// TIA Portal project "Project3" (V15.1)

(* hardware
DEVICE "S7-1200 station_1"  S7-1200 Station
   slot 0: "Rack_0"  S7-1200 Rack  Rack  V1.0
   slot 1: "PLC_1"  CPU 1214C DC/DC/Rly  6ES7 214-1HG40-0XB0  V4.2
*)

// ===== PLC "PLC_1"  CPU 1214C DC/DC/Rly =====

VAR_GLOBAL   // PLC tag table "Default tag table"
   "Stop" AT %I0.0 : Bool;
   "Start" AT %I0.1 : Bool;
   "CIKIS" AT %Q0.2 : Bool;
   "Tag_1" AT %Q0.3 : Bool;
END_VAR

ORGANIZATION_BLOCK "Main"   // OB1, LAD, ProgramCycle
TITLE = "Main Program Sweep (Cycle)"
{ S7_Optimized_Access := 'TRUE' }
VERSION : 0.1
   VAR_INPUT
      Initial_Call : Bool;   // Initial call of this OB
      Remanence : Bool;   // =True, if remanent data are available
   END_VAR
BEGIN

REGION Network 1
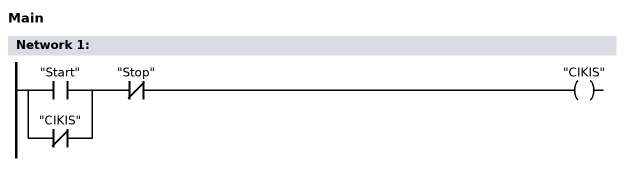
   RUNG wire#powerrail
      Contact( "Start" )
      wire#w1
      I_Contact( "Stop" )
      Coil( "CIKIS" )
   END_RUNG
   RUNG wire#powerrail
      I_Contact( "CIKIS" )
   END_RUNG wire#w1
   // the same network as SCL:
   "CIKIS" := ("Start" OR NOT "CIKIS") AND NOT "Stop";
END_REGION
END_ORGANIZATION_BLOCK